Fanuc KAREL source: kt00438.KL

-- PROVISIONAL review KL for V770-1; original PC SHA256 509672ea202c64b7ff67f2e9245eac4f976c24d8a44f6f1fe8df3f639d722951
-- Incomplete behavior may be omitted. Consult companion uncertainty JSON. Do not deploy.
PROGRAM KT00438
%NOLOCKGROUP
VAR
  I1 : INTEGER
  R2 : REAL
  OUT : BOOLEAN
BEGIN
  -- UNRESOLVED_PC offsets 5-16; opcodes 2E,23
  -- UNRESOLVED_PC offsets 21-32; opcodes 2E,23
  -- UNRESOLVED_PC offsets 37-59; opcodes 21,21,29,64,29,72,23
  -- UNRESOLVED_PC offsets 64-68; opcodes 7F
END KT00438
